FUNCTION_BLOCK FB_Camera
VAR
	_IV3 : BOOL;
END_VAR

METHOD PROTECTED _scanner
VAR_INPUT
	_scanner : BOOL;
END_VAR
END_METHOD

END_FUNCTION_BLOCK

(* stored: Version 1.1.0.1, ProductVersion 3.1.4024.12
   POU FB_Camera: Id {65979892-032e-45c7-85f8-32f178bd09d1}, SpecialFunc None
   Method _scanner: Id {035e3899-2798-4c63-a1c6-9bb0ead59095} *)
